FUNCTION_BLOCK Stage0 (* Template for a Basic Function Block Type *)
  (* Standard: 61499-2 *)
  (* Version 1.0, 2021-06-20, HP *)
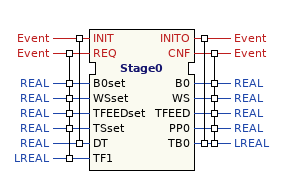
  EVENT_INPUT
    INIT WITH DT; (* Initialization Request *)
    REQ WITH B0set, WSset, TFEEDset, TSset, TF1; (* Normal Execution Request *)
  END_EVENT
  EVENT_OUTPUT
    INITO WITH TB0; (* Initialization Confirm *)
    CNF WITH TB0, PP0, B0, WS, TFEED; (* Execution Confirmation *)
  END_EVENT
  VAR_INPUT
    B0set : REAL; (* Recycle Brine Flow rate (ton/min *)
    WSset : REAL; (* Steam Flow Rate (kg/min) *)
    TFEEDset : REAL; (* Feed Temperature (C) *)
    TSset : REAL; (* Steam Temperature (C) *)
    DT : REAL; (* delta time iteration (s) *)
    TF1 : LREAL; (* Condenser Temperature (C) *)
  END_VAR
  VAR_OUTPUT
    B0 : REAL; (* Recycle Brine Flow Rate (ton/min) *)
    WS : REAL; (* Steam Flow Rate (kg/min) *)
    TFEED : REAL; (* Feed Temperature (C) *)
    PP0 : REAL; (* Pressure of Saturated Steam (atm) *)
    TB0 : LREAL; (* Top Brine Temperature (C) *)
  END_VAR
  VAR
    AB : REAL; (* Internal Variabel *)
    UU : REAL; (* Internal Variabel *)
    TREF : REAL; (* Internal Variabel *)
    AD : REAL; (* Internal Variabel *)
    AHC : REAL; (* Internal Variabel *)
    AHR : REAL; (* Internal Variabel *)
    AS : REAL; (* Internal Variabel *)
    REC : REAL; (* Internal Variabel *)
    WN : REAL; (* Internal Variabel *)
    WN_1 : REAL; (* Internal Variabel *)
    XKN : REAL; (* Internal Variabel *)
    C1 : REAL; (* Internal Variabel *)
    HS : REAL; (* Internal Variabel *)
    G : REAL; (* Internal Variabel *)
    W1 : REAL; (* Internal Variabel *)
    T0 : REAL; (* Internal Variabel *)
    TT : REAL;
    xt : REAL;
    TFREC : REAL; (* Internal Variabel *)
    TS : REAL; (* Internal Variabel *)
    DTS : REAL; (* Internal Variabel *)
    TB0_last : REAL; (* Internal Variabel *)
    USS : REAL; (* Internal Variabel *)
    RHOB : REAL; (* Internal Variabel *)
    CPB0 : REAL; (* Internal Variabel *)
    CPF : REAL; (* Internal Variabel *)
    FMW : REAL; (* Internal Variabel *)
    HLV : REAL; (* Internal Variabel *)
    HLV0 : REAL;
    HV : REAL; (* Internal Variabel *)
    BPR : REAL; (* Internal Variabel *)
    FMC : REAL; (* Internal Variabel *)
    U : REAL; (* Internal Variabel *)
    x : REAL;
    x1 : REAL;
    y : REAL;
    z : REAL;
    b0 : REAL;
    b1 : REAL;
    aa : REAL;
    b2 : REAL;
    b3 : REAL;
    b4 : REAL;
    b5 : REAL;
    b6 : REAL;
    b7 : REAL;
    f0 : REAL;
    ff : REAL;
    JK : REAL;
    PPs : REAL;
    P : REAL;
    HVV : REAL;
    HD : REAL;
    A : REAL; (* Internal Variabel *)
    B : REAL; (* Internal Variabel *)
    C : REAL; (* Internal Variabel *)
    a : REAL;
    p : REAL;
    q : REAL;
    b : REAL;
    l : REAL;
    D1 : REAL; (* Internal Variabel *)
    TC : REAL; (* Internal Variabel *)
    TC1 : REAL;
    PC : REAL; (* Internal Variabel *)
    DTB0 : REAL; (* Internal Variabel *)
    DEN0 : REAL; (* Internal Variabel *)
    DTB1 : REAL; (* Internal Variabel *)
    DENs : REAL; (* Internal Variabel *)
    d : REAL;
    A1 : REAL;
    A2 : REAL;
    A3 : REAL;
    A4 : REAL;
    A5 : REAL;
    A6 : REAL;
    m : REAL;
    n : REAL;
    t1 : REAL;
    t2 : REAL;
    t3 : REAL;
    DELTA67 : REAL;
    DELTA67_last : REAL; (* Internal Variabel *)
  END_VAR
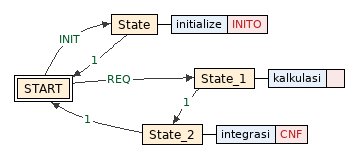
  EC_STATES
    START; (* Initial State *)
    State : initialize -> INITO;
    State_1 : kalkulasi;
    State_2 : integrasi -> CNF;
  END_STATES
  EC_TRANSITIONS
    START TO State := INIT;
    State TO START := 1;
    START TO State_1 := REQ;
    State_1 TO State_2 := 1;
    State_2 TO START := 1;
  END_TRANSITIONS
  ALGORITHM initialize IN ST: (* Initialization algorithm *)
TREF :=273.15;
AB :=57.2727;
AHC :=4069.2;
AHR :=2639.7;
AS :=3225.7;
REC :=0.0;
//TF2:=TF2;

//TFEED :=TFEED1+TREF;
 //TS:=TS1+TREF;
WN :=3.0;
XKN :=0.68;
HS:=0.11;
G :=9.81;
W1 :=0.50;

   //initial condition
TB0   := 366.045551331274;
TFREC := 314.54;
//TS :=TS1;
//DTS := TS-(TF1+TB0)*0.5;
TB0_last :=TB0;
  END_ALGORITHM
  ALGORITHM kalkulasi IN ST: (* perhitungan *)
B0 :=B0set;
WS :=WSset;
TFEED:=TFEEDset+TREF;
TS:=TSset+TREF;
UU := TFEEDset;
U :=UU;

USS :=49.767;
C1 :=0.625;
RHOB :=1032.4; //maassa jenis brine
CPB0 :=1.00; //heatcapacity Brine
CPF :=1.00; //heat capacity feed
FMW :=23654.0;
HLV :=563.7959;
HV :=625.1971;
BPR :=2.192;
FMC :=34736.09;
//US:=USS;
//U :=UU; //feed temp

//////LATENT TS /////
BPR:=0.0;
TT:=(TS-273.15)*1.8+32.0;
TT:=TT-BPR;
T0:=(TT-32.0)/1.8+273.15;
T0:=TS;

 x:=T0*T0;
 y:=80870.0;
 z :=y/x;
 p :=T0*T0*T0;
 x1 :=10.0;
 aa:=T0*(EXPT(x1, z));
b1 :=2641.62/aa;
b2 :=82.546;
b3 :=162460.0/T0;
b4:=0.21828*T0;
b5:=126970.0/T0;
b0:=1.89-b1;
f0:=1.89-b1*(372420/x+2.0);
b6:=b0*b3-2*f0*(b2-b3);
b7:=2*f0*(b4-b5)-b0*b5;
ff:=775.596+0.63296*T0+0.000162467*x;
JK:=log(p);
ff:=ff+(47.3635*JK);

///PRESS TS//
A1 :=3.2437814;
A2:=5.86826*0.001;
A3:=1.1702379*0.00000001;
A4 :=2.1878462*0.001;
A5 :=647.27;
A6 :=218.167;

DTs :=A5-T0;
DENs :=(A1+A2*DTs+A3*DTs*DTs*DTs)/(1+A4*DTs)*DTs/T0;
p:=DENs;
q:=10.0;
PPs :=A6/(EXPT(q, p));

P := PPs;
HV:=(f0*P+b0/2*((P/T0)*(P/T0))*(-b6+b0*(b2-b3+2*b7*((P/T0)*(P/T0)))));
HV:=ff+0.043557*HV;

TC1:=T0-273.15;
HVV:=(2499.15+1.955*TC1-0.001927*TC1*TC1)/4.1868;

 t1:=TT*TT;
 t2:=TT*TT*TT;
 t3:=TT*TT*TT*TT;
HD:=1.0011833*TT-(0.000030833326*t1)-31.92;
HD:=HD+(0.00000004666663*t2)+(0.0000000003333334*t3);

HLV:=HV-HD;

HLV:=HLV*252/0.4536/1000.0;
HLV:=HVV-HD*252/0.4536/1000.0;


HLV0 := HLV;
DTS:=WS*HLV0/USS/AS;

//// state equation
DELTA67:=(B0*(CPF*TF1-CPB0*TB0)*1000.0+USS*AS*DTS)/FMC/CPF;

///  Calculate the physical properties
A :=3.2437814;
B :=5.86826*0.001;
C :=1.1702379*0.00000001;
D1 :=2.1878462*0.001;
TC :=647.27;
PC :=218.167;

DTB0 :=TC-TB0;
DEN0 :=(A+B*DTB0+C*DTB0*DTB0*DTB0)/(1+D1*DTB0)*DTB0/TB0;
b:=DEN0;
a:=10.0;
PP0 :=PC/(EXPT(a, b));
  END_ALGORITHM
  ALGORITHM integrasi IN ST: (* algoritma integrasi *)
B0 :=B0set;
WS :=WSset;
TFEED:=TFEEDset+TREF;
//integrasi

TB0 :=(DELTA67 + DELTA67_last)*0.5*DT + TB0_last;
DELTA67_last :=DELTA67;
TB0_last:=TB0;
  END_ALGORITHM
END_FUNCTION_BLOCK
